TYPE ST_System_MVKW_Stellwert :
STRUCT
	Anford_Stellventil		: BOOL;
	Anford_Pumpe		: BOOL;
	Anford_Kompressor	: BOOL;
END_STRUCT
END_TYPE

(* stored: Version 1.1.0.1, ProductVersion 3.1.4024.9
   DUT ST_System_MVKW_Stellwert: Id {881d1f96-f815-4de6-b7dc-f2883d7c1228} *)
